PROGRAM PRG_SDS_Y_EPS
VAR
    bInit 		: BOOL := TRUE;
    bFullRange	: BOOL;
    nIndex 		: uint;
    nEPSIndex 	: uint;

    fSDS_Z_ENC 	: LREAL;
    fSDS_RY 	: LREAL;
    fSDS_Y 		: LREAL;
    fRCC_Y 		: LREAL;

    fbEPS		: FB_EPS;

END_VAR

// SDS Y EPS
IF bInit THEN
    // Set Inital Values
    aSDS_Y_EPS[1].fBwd_Limits := 20;
    aSDS_Y_EPS[1].fFwd_Limits := 45;

    aSDS_Y_EPS[2].fBwd_Limits := 37.5;
    aSDS_Y_EPS[2].fFwd_Limits := 38.5;

    aSDS_Y_EPS[3].fBwd_Limits := 30;
    aSDS_Y_EPS[3].fFwd_Limits := 38.5;

    aSDS_Y_EPS[4].fBwd_Limits := 30;
    aSDS_Y_EPS[4].fFwd_Limits := 35;

    aSDS_Y_EPS[5].fBwd_Limits := 30;
    aSDS_Y_EPS[5].fFwd_Limits := 45;


    bInit := FALSE;
END_IF

// Encoder / position values
fSDS_Z_ENC :=  M36.stAxisStatus.fActPosition;
fSDS_RY := M19.stAxisStatus.fActPosition;
fSDS_Y  := M17.stAxisStatus.fActPosition;
fRCC_Y  := M38.stAxisStatus.fActPosition;

// Set EPS conditions
fbEPS(eps:= aSDS_Y_EPS[2].stEPS);
fbEPS.setDescription('SDS_Z_ENC in [0,400]');
fbEPS.setBit(0, F_InRange(fSDS_Z_ENC, 0, 400));

fbEPS(eps:= aSDS_Y_EPS[3].stEPS);
fbEPS.setDescription('SDS_Z_ENC in [400,420];SDS_RY in [-5,5]');
fbEPS.setBit(0, F_InRange(fSDS_Z_ENC, 400, 420));
fbEPS.setBit(1, F_InRange(fSDS_RY, -5, 5));

fbEPS(eps:= aSDS_Y_EPS[4].stEPS);
fbEPS.setDescription('SDS_Z_ENC in [400,495];SDS_RY in [-100,-5]');
fbEPS.setBit(0, F_InRange(fSDS_Z_ENC, 400, 495));
fbEPS.setBit(1, F_InRange(fSDS_RY, -100, -5));

fbEPS(eps:= aSDS_Y_EPS[5].stEPS);
fbEPS.setDescription('SDS_Z_ENC in [495,510];(SDS_Y - RCC >= 36');
fbEPS.setBit(0, F_InRange(fSDS_Z_ENC, 495, 510));
fbEPS.setBit(1, (fSDS_Y - fRCC_Y) >= 36);


bFullRange := (NOT aSDS_Y_EPS[2].stEPS.bEPS_OK) AND (NOT aSDS_Y_EPS[3].stEPS.bEPS_OK) AND(NOT aSDS_Y_EPS[4].stEPS.bEPS_OK) AND (NOT aSDS_Y_EPS[5].stEPS.bEPS_OK);
fbEPS(eps:= aSDS_Y_EPS[1].stEPS);
fbEPS.setBit(0, bFullRange); // FULL RANGE

F_CheckEPSArray(stMotor:=M17, aEPSLimits:=aSDS_Y_EPS, 1 ,5);

END_PROGRAM

(* stored: Version 1.1.0.1, ProductVersion 3.1.4022.18
   POU PRG_SDS_Y_EPS: Id {1d694921-86bf-430a-8dcf-197fd1ce1485}, SpecialFunc None *)
